(* Logix 5000 project; controller R1USB70001_CWRU_Scenario_Gen_20111116 vendor 1 type 14 code 54 rev 19.11; software revision 19.01; part 7 of 9 *)
(* tags used below, declared in another part *)
   EditScenario : EditScenarioPub;
   HMI : HMIPub;
   HMI_Intfc_Read_Buffer : DINT[40];
(* MainProgram, continued *)

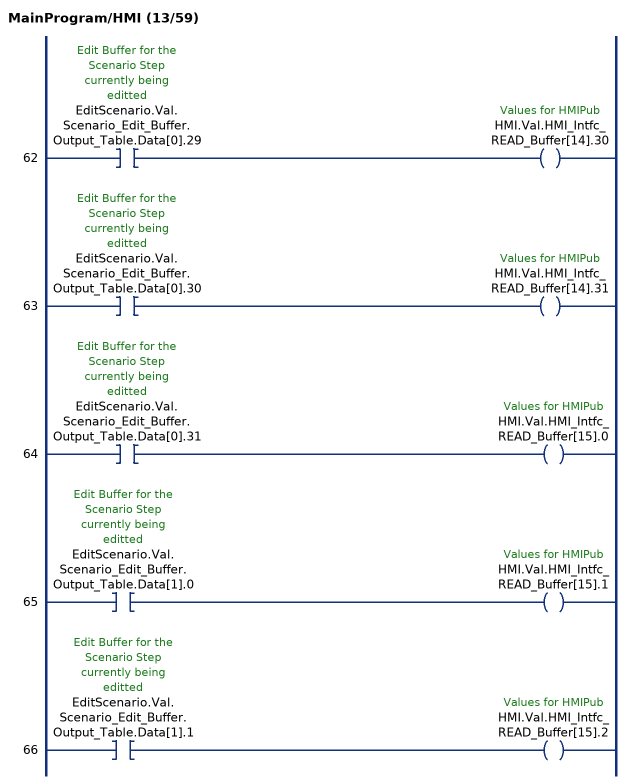
   62: XIC(EditScenario.Val.Scenario_Edit_Buffer.Output_Table.Data[0].29)OTE(HMI.Val.HMI_Intfc_READ_Buffer[14].30);
   63: XIC(EditScenario.Val.Scenario_Edit_Buffer.Output_Table.Data[0].30)OTE(HMI.Val.HMI_Intfc_READ_Buffer[14].31);
   64: XIC(EditScenario.Val.Scenario_Edit_Buffer.Output_Table.Data[0].31)OTE(HMI.Val.HMI_Intfc_READ_Buffer[15].0);
   65: XIC(EditScenario.Val.Scenario_Edit_Buffer.Output_Table.Data[1].0)OTE(HMI.Val.HMI_Intfc_READ_Buffer[15].1);
   66: XIC(EditScenario.Val.Scenario_Edit_Buffer.Output_Table.Data[1].1)OTE(HMI.Val.HMI_Intfc_READ_Buffer[15].2);
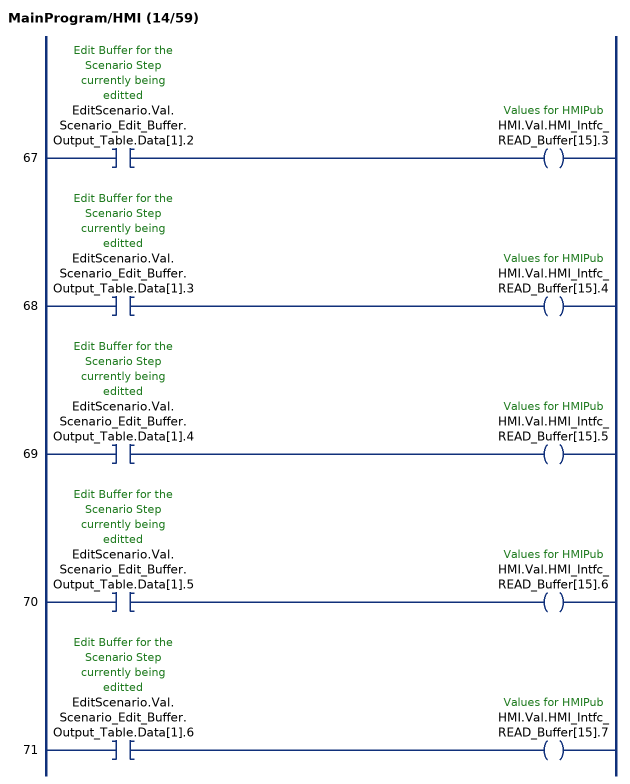
   67: XIC(EditScenario.Val.Scenario_Edit_Buffer.Output_Table.Data[1].2)OTE(HMI.Val.HMI_Intfc_READ_Buffer[15].3);
   68: XIC(EditScenario.Val.Scenario_Edit_Buffer.Output_Table.Data[1].3)OTE(HMI.Val.HMI_Intfc_READ_Buffer[15].4);
   69: XIC(EditScenario.Val.Scenario_Edit_Buffer.Output_Table.Data[1].4)OTE(HMI.Val.HMI_Intfc_READ_Buffer[15].5);
   70: XIC(EditScenario.Val.Scenario_Edit_Buffer.Output_Table.Data[1].5)OTE(HMI.Val.HMI_Intfc_READ_Buffer[15].6);
   71: XIC(EditScenario.Val.Scenario_Edit_Buffer.Output_Table.Data[1].6)OTE(HMI.Val.HMI_Intfc_READ_Buffer[15].7);
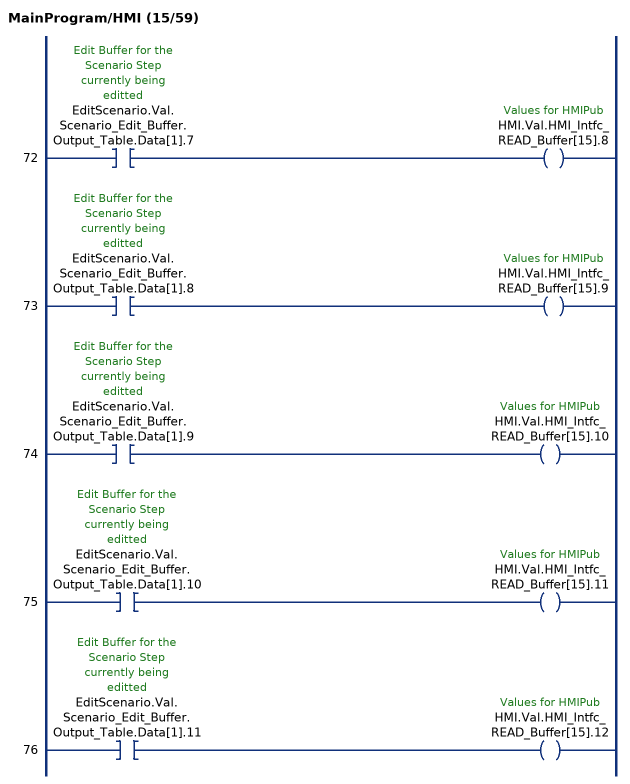
   72: XIC(EditScenario.Val.Scenario_Edit_Buffer.Output_Table.Data[1].7)OTE(HMI.Val.HMI_Intfc_READ_Buffer[15].8);
   73: XIC(EditScenario.Val.Scenario_Edit_Buffer.Output_Table.Data[1].8)OTE(HMI.Val.HMI_Intfc_READ_Buffer[15].9);
   74: XIC(EditScenario.Val.Scenario_Edit_Buffer.Output_Table.Data[1].9)OTE(HMI.Val.HMI_Intfc_READ_Buffer[15].10);
   75: XIC(EditScenario.Val.Scenario_Edit_Buffer.Output_Table.Data[1].10)OTE(HMI.Val.HMI_Intfc_READ_Buffer[15].11);
   76: XIC(EditScenario.Val.Scenario_Edit_Buffer.Output_Table.Data[1].11)OTE(HMI.Val.HMI_Intfc_READ_Buffer[15].12);
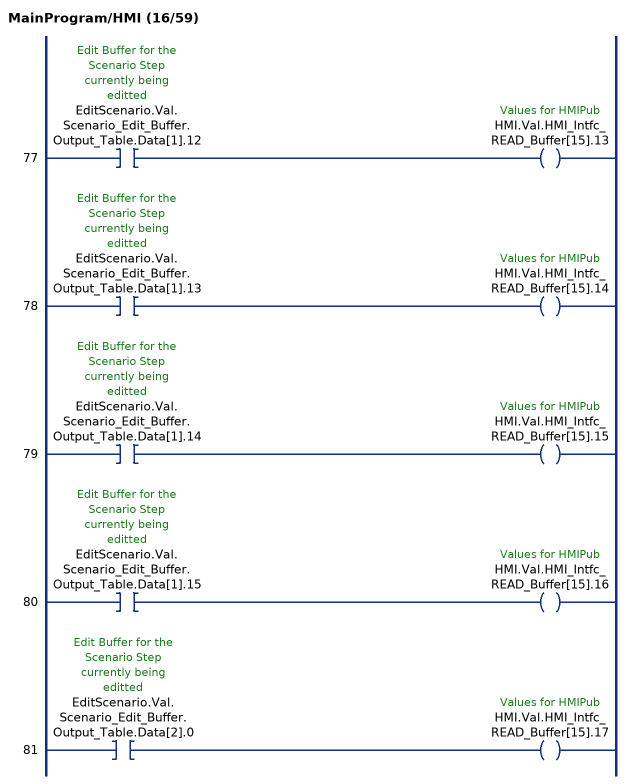
   77: XIC(EditScenario.Val.Scenario_Edit_Buffer.Output_Table.Data[1].12)OTE(HMI.Val.HMI_Intfc_READ_Buffer[15].13);
   78: XIC(EditScenario.Val.Scenario_Edit_Buffer.Output_Table.Data[1].13)OTE(HMI.Val.HMI_Intfc_READ_Buffer[15].14);
   79: XIC(EditScenario.Val.Scenario_Edit_Buffer.Output_Table.Data[1].14)OTE(HMI.Val.HMI_Intfc_READ_Buffer[15].15);
   80: XIC(EditScenario.Val.Scenario_Edit_Buffer.Output_Table.Data[1].15)OTE(HMI.Val.HMI_Intfc_READ_Buffer[15].16);
   81: XIC(EditScenario.Val.Scenario_Edit_Buffer.Output_Table.Data[2].0)OTE(HMI.Val.HMI_Intfc_READ_Buffer[15].17);
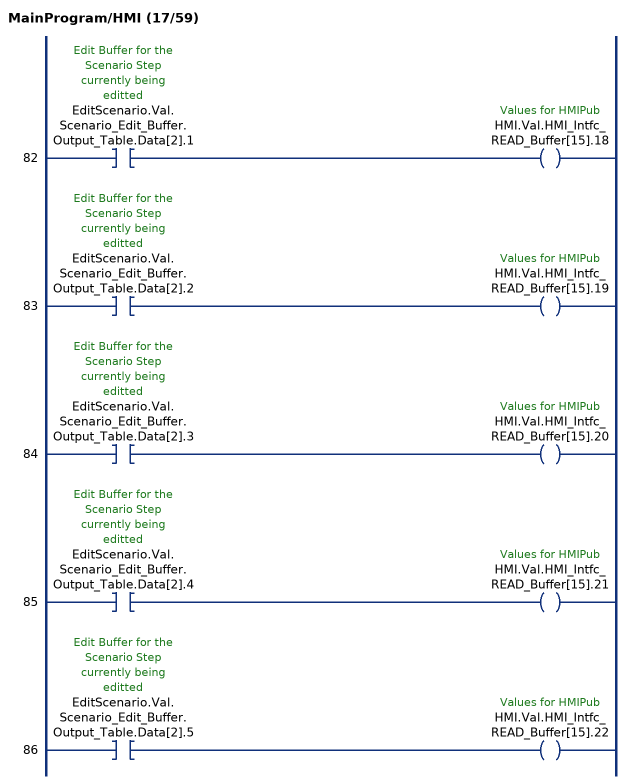
   82: XIC(EditScenario.Val.Scenario_Edit_Buffer.Output_Table.Data[2].1)OTE(HMI.Val.HMI_Intfc_READ_Buffer[15].18);
   83: XIC(EditScenario.Val.Scenario_Edit_Buffer.Output_Table.Data[2].2)OTE(HMI.Val.HMI_Intfc_READ_Buffer[15].19);
   84: XIC(EditScenario.Val.Scenario_Edit_Buffer.Output_Table.Data[2].3)OTE(HMI.Val.HMI_Intfc_READ_Buffer[15].20);
   85: XIC(EditScenario.Val.Scenario_Edit_Buffer.Output_Table.Data[2].4)OTE(HMI.Val.HMI_Intfc_READ_Buffer[15].21);
   86: XIC(EditScenario.Val.Scenario_Edit_Buffer.Output_Table.Data[2].5)OTE(HMI.Val.HMI_Intfc_READ_Buffer[15].22);
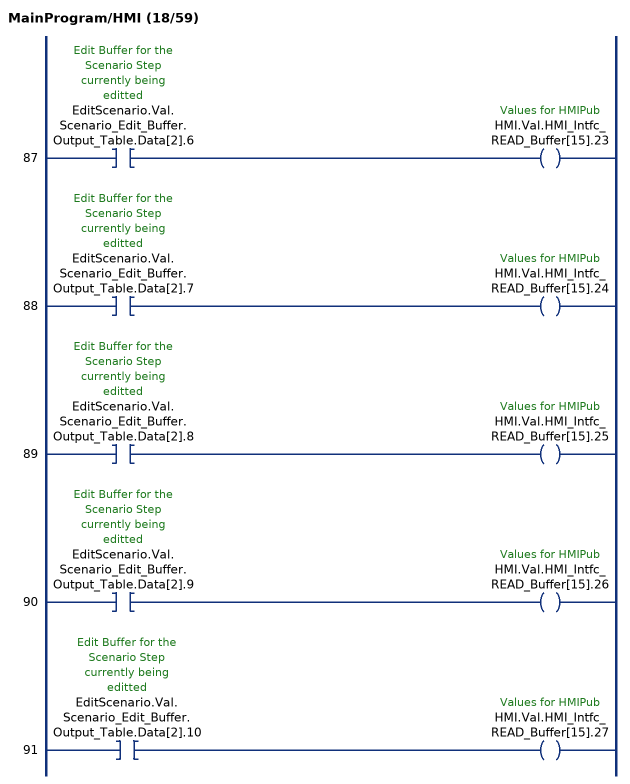
   87: XIC(EditScenario.Val.Scenario_Edit_Buffer.Output_Table.Data[2].6)OTE(HMI.Val.HMI_Intfc_READ_Buffer[15].23);
   88: XIC(EditScenario.Val.Scenario_Edit_Buffer.Output_Table.Data[2].7)OTE(HMI.Val.HMI_Intfc_READ_Buffer[15].24);
   89: XIC(EditScenario.Val.Scenario_Edit_Buffer.Output_Table.Data[2].8)OTE(HMI.Val.HMI_Intfc_READ_Buffer[15].25);
   90: XIC(EditScenario.Val.Scenario_Edit_Buffer.Output_Table.Data[2].9)OTE(HMI.Val.HMI_Intfc_READ_Buffer[15].26);
   91: XIC(EditScenario.Val.Scenario_Edit_Buffer.Output_Table.Data[2].10)OTE(HMI.Val.HMI_Intfc_READ_Buffer[15].27);
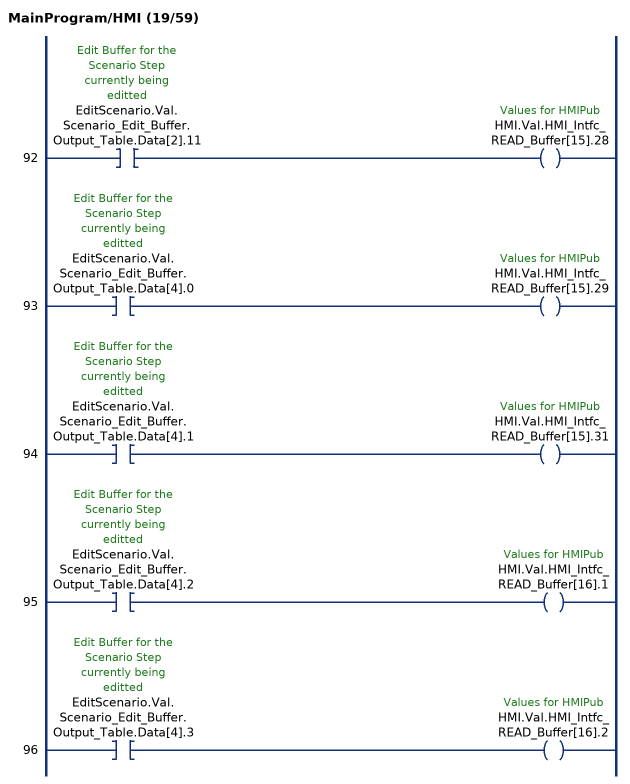
   92: XIC(EditScenario.Val.Scenario_Edit_Buffer.Output_Table.Data[2].11)OTE(HMI.Val.HMI_Intfc_READ_Buffer[15].28);
   93: XIC(EditScenario.Val.Scenario_Edit_Buffer.Output_Table.Data[4].0)OTE(HMI.Val.HMI_Intfc_READ_Buffer[15].29);
   94: XIC(EditScenario.Val.Scenario_Edit_Buffer.Output_Table.Data[4].1)OTE(HMI.Val.HMI_Intfc_READ_Buffer[15].31);
   95: XIC(EditScenario.Val.Scenario_Edit_Buffer.Output_Table.Data[4].2)OTE(HMI.Val.HMI_Intfc_READ_Buffer[16].1);
   96: XIC(EditScenario.Val.Scenario_Edit_Buffer.Output_Table.Data[4].3)OTE(HMI.Val.HMI_Intfc_READ_Buffer[16].2);
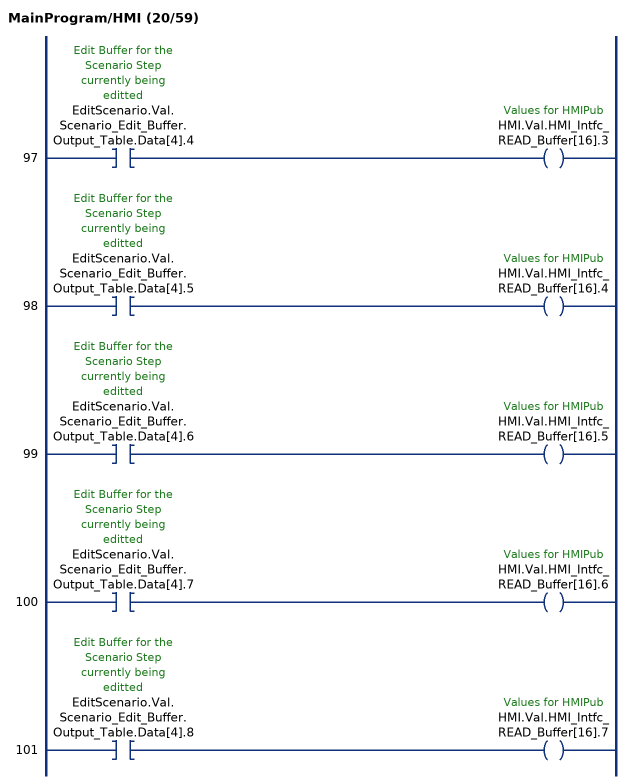
   97: XIC(EditScenario.Val.Scenario_Edit_Buffer.Output_Table.Data[4].4)OTE(HMI.Val.HMI_Intfc_READ_Buffer[16].3);
   98: XIC(EditScenario.Val.Scenario_Edit_Buffer.Output_Table.Data[4].5)OTE(HMI.Val.HMI_Intfc_READ_Buffer[16].4);
   99: XIC(EditScenario.Val.Scenario_Edit_Buffer.Output_Table.Data[4].6)OTE(HMI.Val.HMI_Intfc_READ_Buffer[16].5);
   100: XIC(EditScenario.Val.Scenario_Edit_Buffer.Output_Table.Data[4].7)OTE(HMI.Val.HMI_Intfc_READ_Buffer[16].6);
   101: XIC(EditScenario.Val.Scenario_Edit_Buffer.Output_Table.Data[4].8)OTE(HMI.Val.HMI_Intfc_READ_Buffer[16].7);
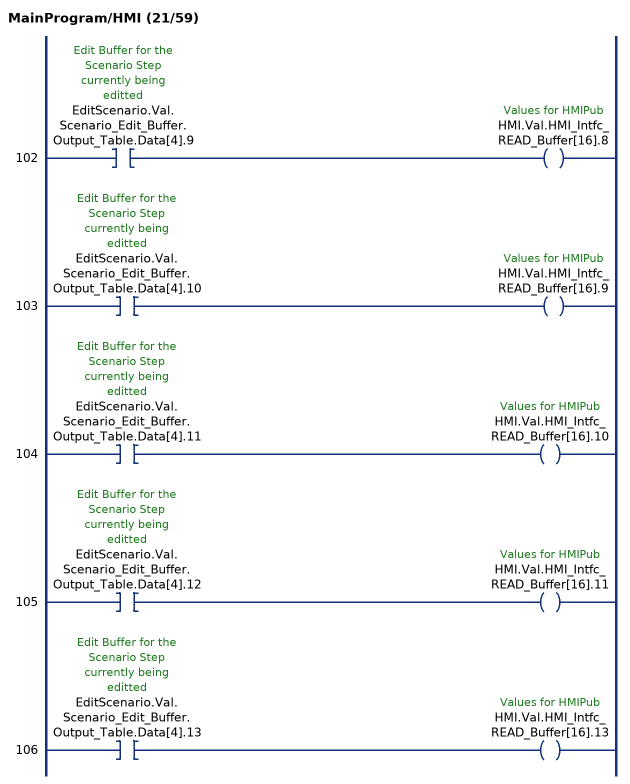
   102: XIC(EditScenario.Val.Scenario_Edit_Buffer.Output_Table.Data[4].9)OTE(HMI.Val.HMI_Intfc_READ_Buffer[16].8);
   103: XIC(EditScenario.Val.Scenario_Edit_Buffer.Output_Table.Data[4].10)OTE(HMI.Val.HMI_Intfc_READ_Buffer[16].9);
   104: XIC(EditScenario.Val.Scenario_Edit_Buffer.Output_Table.Data[4].11)OTE(HMI.Val.HMI_Intfc_READ_Buffer[16].10);
   105: XIC(EditScenario.Val.Scenario_Edit_Buffer.Output_Table.Data[4].12)OTE(HMI.Val.HMI_Intfc_READ_Buffer[16].11);
   106: XIC(EditScenario.Val.Scenario_Edit_Buffer.Output_Table.Data[4].13)OTE(HMI.Val.HMI_Intfc_READ_Buffer[16].13);
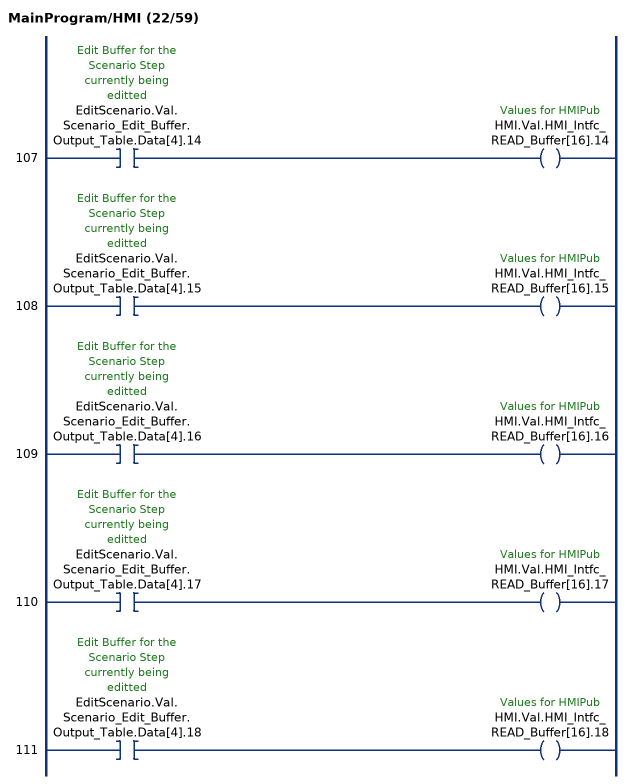
   107: XIC(EditScenario.Val.Scenario_Edit_Buffer.Output_Table.Data[4].14)OTE(HMI.Val.HMI_Intfc_READ_Buffer[16].14);
   108: XIC(EditScenario.Val.Scenario_Edit_Buffer.Output_Table.Data[4].15)OTE(HMI.Val.HMI_Intfc_READ_Buffer[16].15);
   109: XIC(EditScenario.Val.Scenario_Edit_Buffer.Output_Table.Data[4].16)OTE(HMI.Val.HMI_Intfc_READ_Buffer[16].16);
   110: XIC(EditScenario.Val.Scenario_Edit_Buffer.Output_Table.Data[4].17)OTE(HMI.Val.HMI_Intfc_READ_Buffer[16].17);
   111: XIC(EditScenario.Val.Scenario_Edit_Buffer.Output_Table.Data[4].18)OTE(HMI.Val.HMI_Intfc_READ_Buffer[16].18);
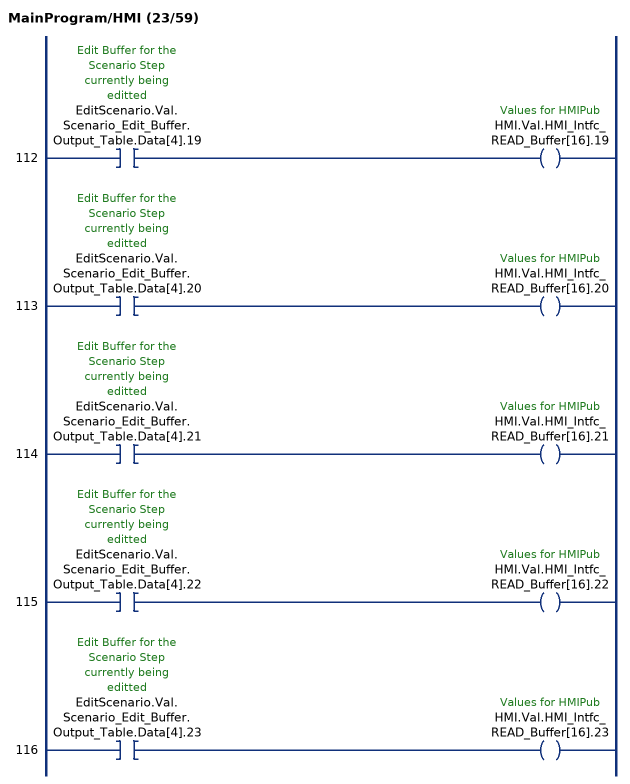
   112: XIC(EditScenario.Val.Scenario_Edit_Buffer.Output_Table.Data[4].19)OTE(HMI.Val.HMI_Intfc_READ_Buffer[16].19);
   113: XIC(EditScenario.Val.Scenario_Edit_Buffer.Output_Table.Data[4].20)OTE(HMI.Val.HMI_Intfc_READ_Buffer[16].20);
   114: XIC(EditScenario.Val.Scenario_Edit_Buffer.Output_Table.Data[4].21)OTE(HMI.Val.HMI_Intfc_READ_Buffer[16].21);
   115: XIC(EditScenario.Val.Scenario_Edit_Buffer.Output_Table.Data[4].22)OTE(HMI.Val.HMI_Intfc_READ_Buffer[16].22);
   116: XIC(EditScenario.Val.Scenario_Edit_Buffer.Output_Table.Data[4].23)OTE(HMI.Val.HMI_Intfc_READ_Buffer[16].23);
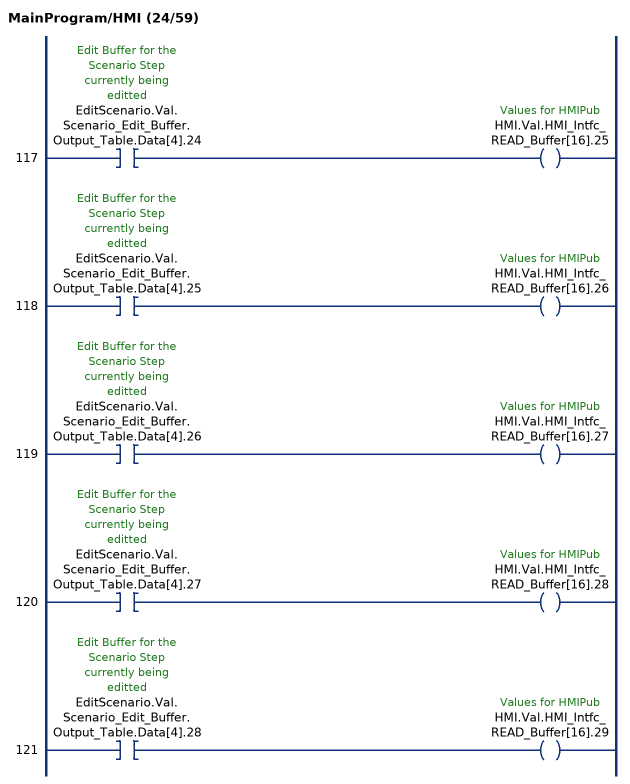
   117: XIC(EditScenario.Val.Scenario_Edit_Buffer.Output_Table.Data[4].24)OTE(HMI.Val.HMI_Intfc_READ_Buffer[16].25);
   118: XIC(EditScenario.Val.Scenario_Edit_Buffer.Output_Table.Data[4].25)OTE(HMI.Val.HMI_Intfc_READ_Buffer[16].26);
   119: XIC(EditScenario.Val.Scenario_Edit_Buffer.Output_Table.Data[4].26)OTE(HMI.Val.HMI_Intfc_READ_Buffer[16].27);
   120: XIC(EditScenario.Val.Scenario_Edit_Buffer.Output_Table.Data[4].27)OTE(HMI.Val.HMI_Intfc_READ_Buffer[16].28);
   121: XIC(EditScenario.Val.Scenario_Edit_Buffer.Output_Table.Data[4].28)OTE(HMI.Val.HMI_Intfc_READ_Buffer[16].29);
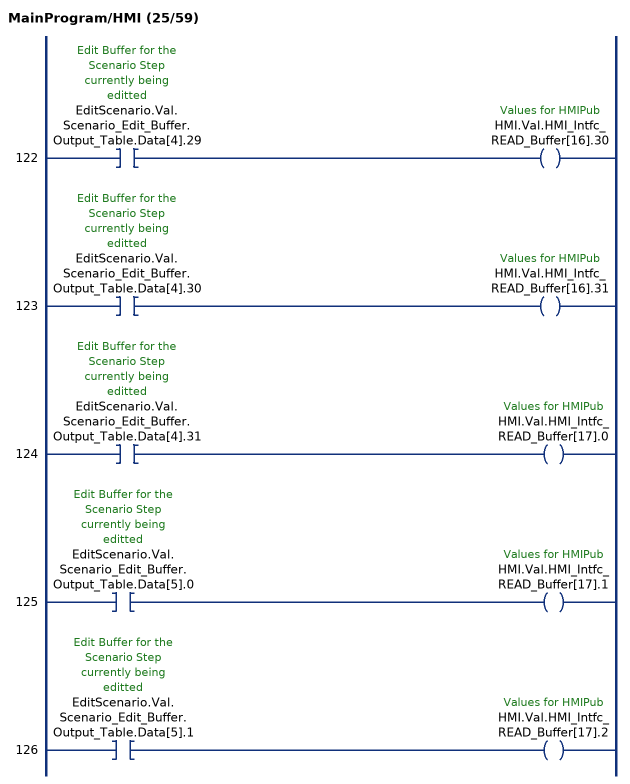
   122: XIC(EditScenario.Val.Scenario_Edit_Buffer.Output_Table.Data[4].29)OTE(HMI.Val.HMI_Intfc_READ_Buffer[16].30);
   123: XIC(EditScenario.Val.Scenario_Edit_Buffer.Output_Table.Data[4].30)OTE(HMI.Val.HMI_Intfc_READ_Buffer[16].31);
   124: XIC(EditScenario.Val.Scenario_Edit_Buffer.Output_Table.Data[4].31)OTE(HMI.Val.HMI_Intfc_READ_Buffer[17].0);
   125: XIC(EditScenario.Val.Scenario_Edit_Buffer.Output_Table.Data[5].0)OTE(HMI.Val.HMI_Intfc_READ_Buffer[17].1);
   126: XIC(EditScenario.Val.Scenario_Edit_Buffer.Output_Table.Data[5].1)OTE(HMI.Val.HMI_Intfc_READ_Buffer[17].2);
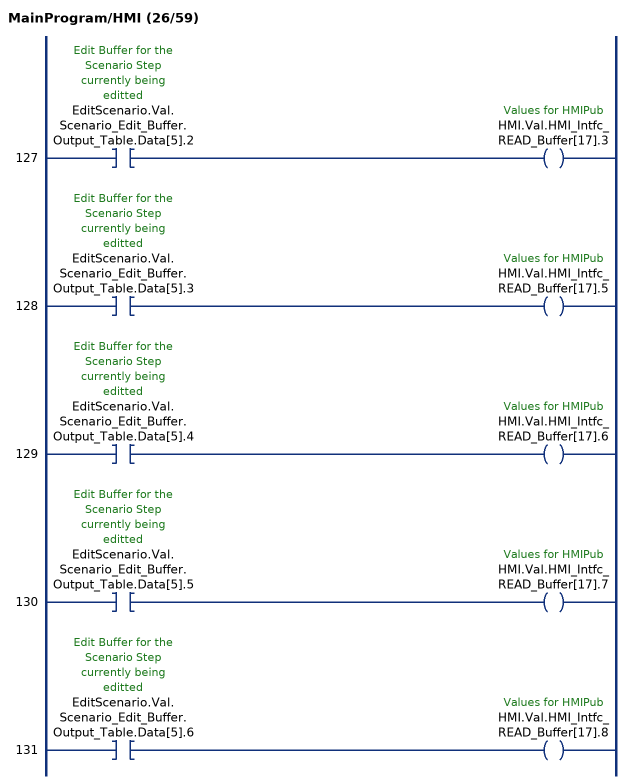
   127: XIC(EditScenario.Val.Scenario_Edit_Buffer.Output_Table.Data[5].2)OTE(HMI.Val.HMI_Intfc_READ_Buffer[17].3);
   128: XIC(EditScenario.Val.Scenario_Edit_Buffer.Output_Table.Data[5].3)OTE(HMI.Val.HMI_Intfc_READ_Buffer[17].5);
   129: XIC(EditScenario.Val.Scenario_Edit_Buffer.Output_Table.Data[5].4)OTE(HMI.Val.HMI_Intfc_READ_Buffer[17].6);
   130: XIC(EditScenario.Val.Scenario_Edit_Buffer.Output_Table.Data[5].5)OTE(HMI.Val.HMI_Intfc_READ_Buffer[17].7);
   131: XIC(EditScenario.Val.Scenario_Edit_Buffer.Output_Table.Data[5].6)OTE(HMI.Val.HMI_Intfc_READ_Buffer[17].8);
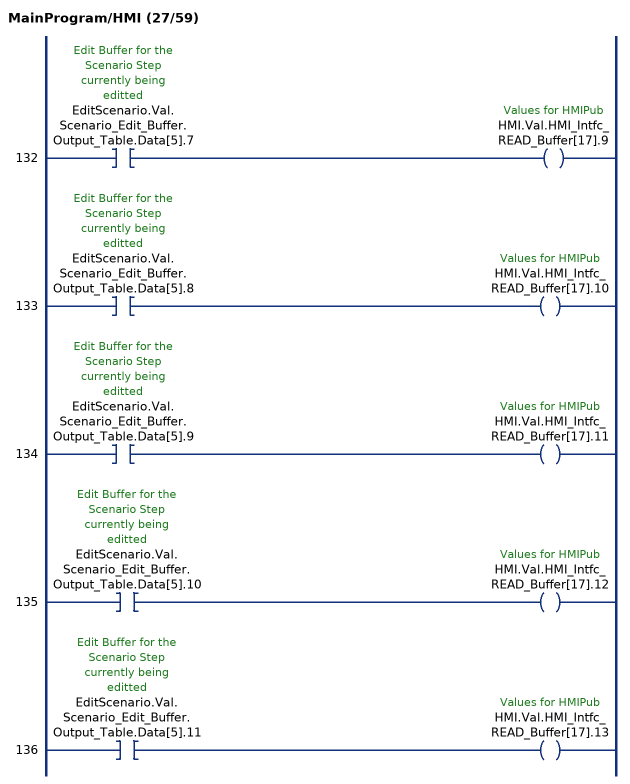
   132: XIC(EditScenario.Val.Scenario_Edit_Buffer.Output_Table.Data[5].7)OTE(HMI.Val.HMI_Intfc_READ_Buffer[17].9);
   133: XIC(EditScenario.Val.Scenario_Edit_Buffer.Output_Table.Data[5].8)OTE(HMI.Val.HMI_Intfc_READ_Buffer[17].10);
   134: XIC(EditScenario.Val.Scenario_Edit_Buffer.Output_Table.Data[5].9)OTE(HMI.Val.HMI_Intfc_READ_Buffer[17].11);
   135: XIC(EditScenario.Val.Scenario_Edit_Buffer.Output_Table.Data[5].10)OTE(HMI.Val.HMI_Intfc_READ_Buffer[17].12);
   136: XIC(EditScenario.Val.Scenario_Edit_Buffer.Output_Table.Data[5].11)OTE(HMI.Val.HMI_Intfc_READ_Buffer[17].13);
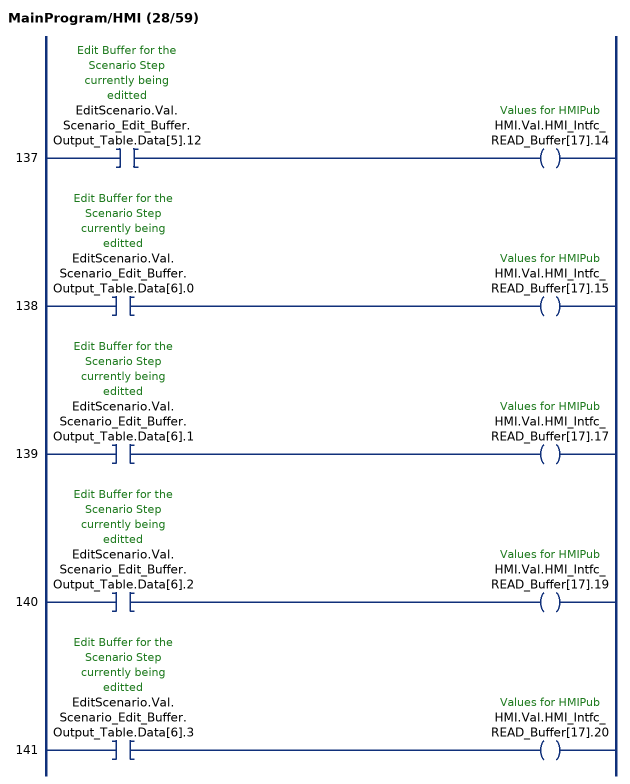
   137: XIC(EditScenario.Val.Scenario_Edit_Buffer.Output_Table.Data[5].12)OTE(HMI.Val.HMI_Intfc_READ_Buffer[17].14);
   138: XIC(EditScenario.Val.Scenario_Edit_Buffer.Output_Table.Data[6].0)OTE(HMI.Val.HMI_Intfc_READ_Buffer[17].15);
   139: XIC(EditScenario.Val.Scenario_Edit_Buffer.Output_Table.Data[6].1)OTE(HMI.Val.HMI_Intfc_READ_Buffer[17].17);
   140: XIC(EditScenario.Val.Scenario_Edit_Buffer.Output_Table.Data[6].2)OTE(HMI.Val.HMI_Intfc_READ_Buffer[17].19);
   141: XIC(EditScenario.Val.Scenario_Edit_Buffer.Output_Table.Data[6].3)OTE(HMI.Val.HMI_Intfc_READ_Buffer[17].20);
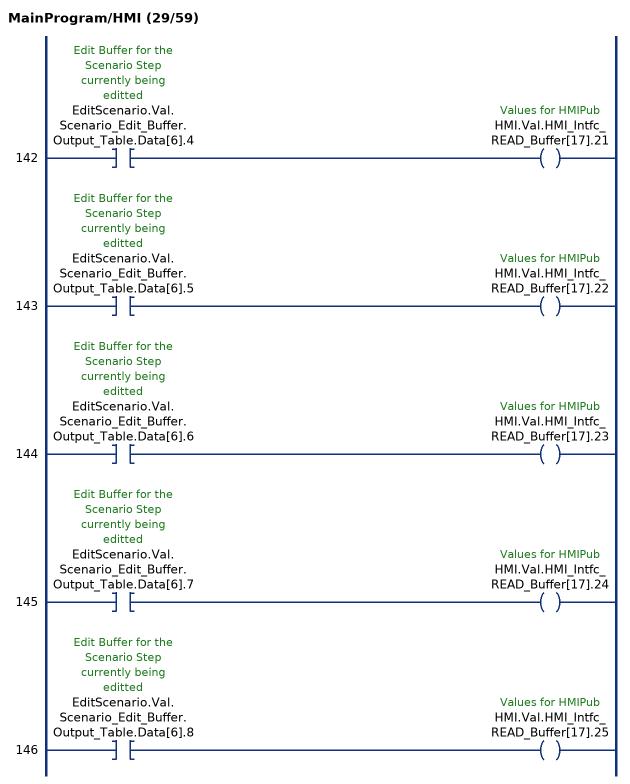
   142: XIC(EditScenario.Val.Scenario_Edit_Buffer.Output_Table.Data[6].4)OTE(HMI.Val.HMI_Intfc_READ_Buffer[17].21);
   143: XIC(EditScenario.Val.Scenario_Edit_Buffer.Output_Table.Data[6].5)OTE(HMI.Val.HMI_Intfc_READ_Buffer[17].22);
   144: XIC(EditScenario.Val.Scenario_Edit_Buffer.Output_Table.Data[6].6)OTE(HMI.Val.HMI_Intfc_READ_Buffer[17].23);
   145: XIC(EditScenario.Val.Scenario_Edit_Buffer.Output_Table.Data[6].7)OTE(HMI.Val.HMI_Intfc_READ_Buffer[17].24);
   146: XIC(EditScenario.Val.Scenario_Edit_Buffer.Output_Table.Data[6].8)OTE(HMI.Val.HMI_Intfc_READ_Buffer[17].25);
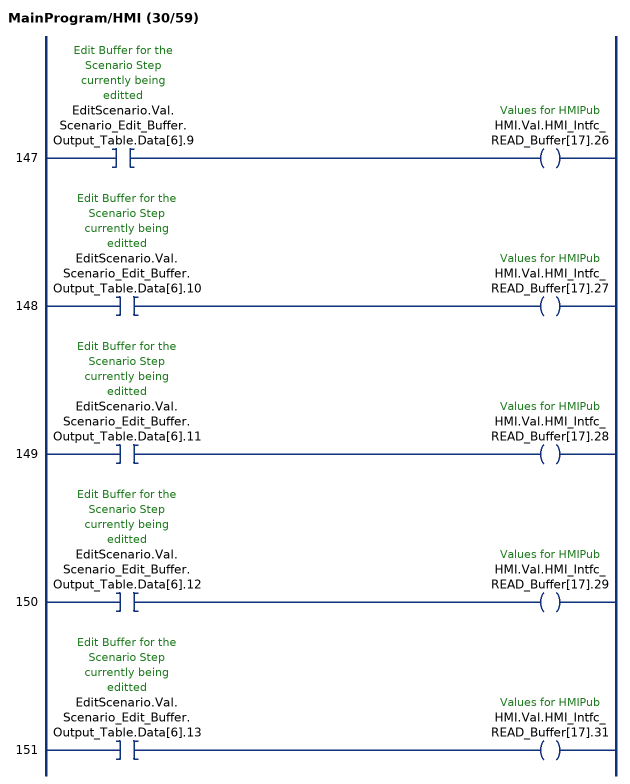
   147: XIC(EditScenario.Val.Scenario_Edit_Buffer.Output_Table.Data[6].9)OTE(HMI.Val.HMI_Intfc_READ_Buffer[17].26);
   148: XIC(EditScenario.Val.Scenario_Edit_Buffer.Output_Table.Data[6].10)OTE(HMI.Val.HMI_Intfc_READ_Buffer[17].27);
   149: XIC(EditScenario.Val.Scenario_Edit_Buffer.Output_Table.Data[6].11)OTE(HMI.Val.HMI_Intfc_READ_Buffer[17].28);
   150: XIC(EditScenario.Val.Scenario_Edit_Buffer.Output_Table.Data[6].12)OTE(HMI.Val.HMI_Intfc_READ_Buffer[17].29);
   151: XIC(EditScenario.Val.Scenario_Edit_Buffer.Output_Table.Data[6].13)OTE(HMI.Val.HMI_Intfc_READ_Buffer[17].31);
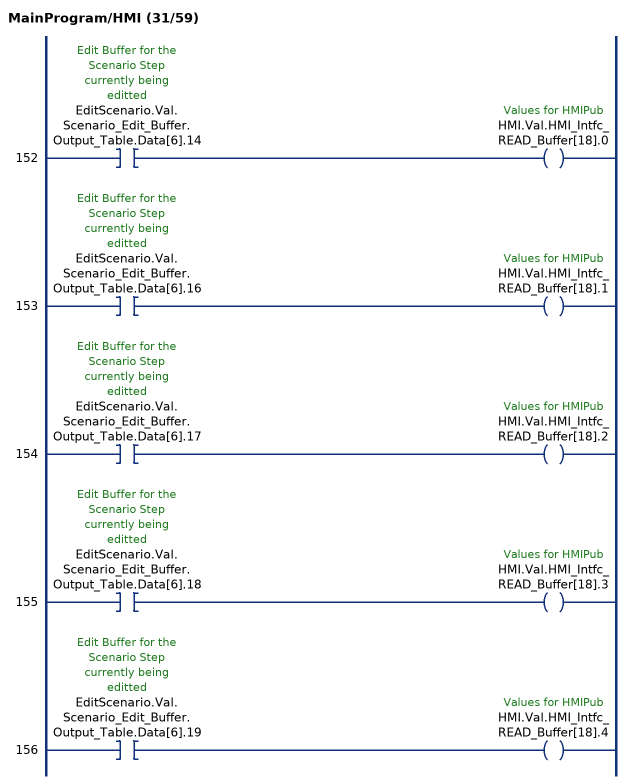
   152: XIC(EditScenario.Val.Scenario_Edit_Buffer.Output_Table.Data[6].14)OTE(HMI.Val.HMI_Intfc_READ_Buffer[18].0);
   153: XIC(EditScenario.Val.Scenario_Edit_Buffer.Output_Table.Data[6].16)OTE(HMI.Val.HMI_Intfc_READ_Buffer[18].1);
   154: XIC(EditScenario.Val.Scenario_Edit_Buffer.Output_Table.Data[6].17)OTE(HMI.Val.HMI_Intfc_READ_Buffer[18].2);
   155: XIC(EditScenario.Val.Scenario_Edit_Buffer.Output_Table.Data[6].18)OTE(HMI.Val.HMI_Intfc_READ_Buffer[18].3);
   156: XIC(EditScenario.Val.Scenario_Edit_Buffer.Output_Table.Data[6].19)OTE(HMI.Val.HMI_Intfc_READ_Buffer[18].4);
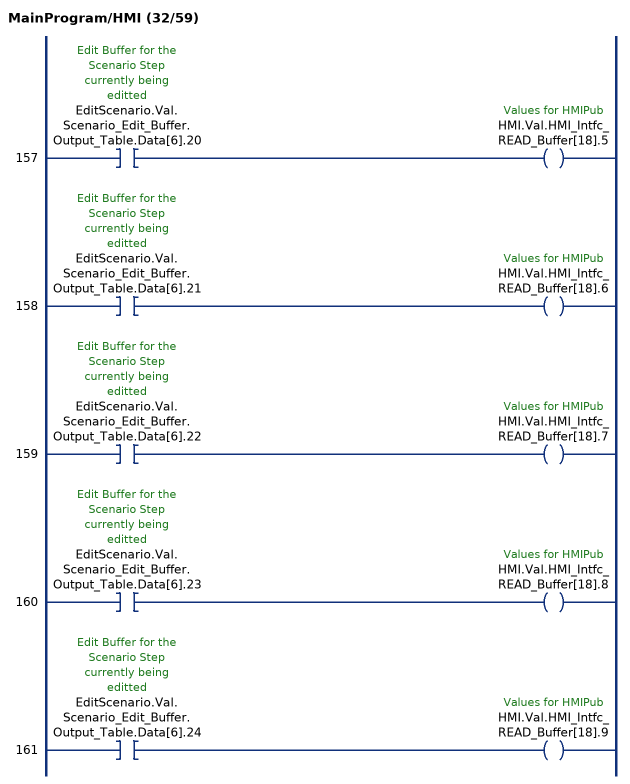
   157: XIC(EditScenario.Val.Scenario_Edit_Buffer.Output_Table.Data[6].20)OTE(HMI.Val.HMI_Intfc_READ_Buffer[18].5);
   158: XIC(EditScenario.Val.Scenario_Edit_Buffer.Output_Table.Data[6].21)OTE(HMI.Val.HMI_Intfc_READ_Buffer[18].6);
   159: XIC(EditScenario.Val.Scenario_Edit_Buffer.Output_Table.Data[6].22)OTE(HMI.Val.HMI_Intfc_READ_Buffer[18].7);
   160: XIC(EditScenario.Val.Scenario_Edit_Buffer.Output_Table.Data[6].23)OTE(HMI.Val.HMI_Intfc_READ_Buffer[18].8);
   161: XIC(EditScenario.Val.Scenario_Edit_Buffer.Output_Table.Data[6].24)OTE(HMI.Val.HMI_Intfc_READ_Buffer[18].9);
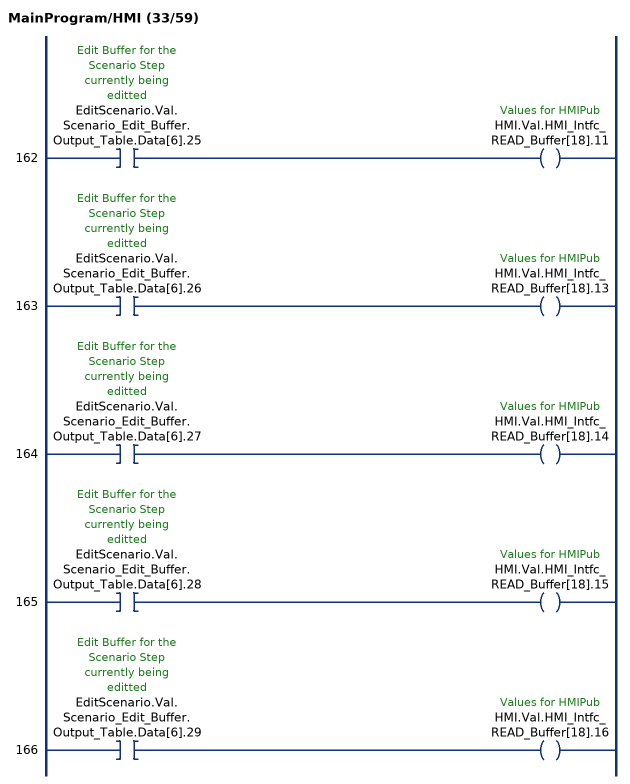
   162: XIC(EditScenario.Val.Scenario_Edit_Buffer.Output_Table.Data[6].25)OTE(HMI.Val.HMI_Intfc_READ_Buffer[18].11);
   163: XIC(EditScenario.Val.Scenario_Edit_Buffer.Output_Table.Data[6].26)OTE(HMI.Val.HMI_Intfc_READ_Buffer[18].13);
   164: XIC(EditScenario.Val.Scenario_Edit_Buffer.Output_Table.Data[6].27)OTE(HMI.Val.HMI_Intfc_READ_Buffer[18].14);
   165: XIC(EditScenario.Val.Scenario_Edit_Buffer.Output_Table.Data[6].28)OTE(HMI.Val.HMI_Intfc_READ_Buffer[18].15);
   166: XIC(EditScenario.Val.Scenario_Edit_Buffer.Output_Table.Data[6].29)OTE(HMI.Val.HMI_Intfc_READ_Buffer[18].16);
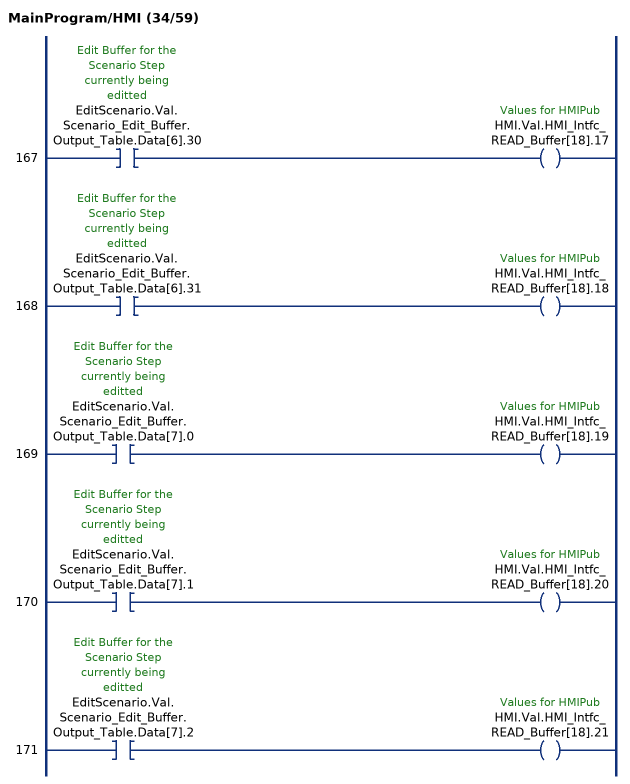
   167: XIC(EditScenario.Val.Scenario_Edit_Buffer.Output_Table.Data[6].30)OTE(HMI.Val.HMI_Intfc_READ_Buffer[18].17);
   168: XIC(EditScenario.Val.Scenario_Edit_Buffer.Output_Table.Data[6].31)OTE(HMI.Val.HMI_Intfc_READ_Buffer[18].18);
   169: XIC(EditScenario.Val.Scenario_Edit_Buffer.Output_Table.Data[7].0)OTE(HMI.Val.HMI_Intfc_READ_Buffer[18].19);
   170: XIC(EditScenario.Val.Scenario_Edit_Buffer.Output_Table.Data[7].1)OTE(HMI.Val.HMI_Intfc_READ_Buffer[18].20);
   171: XIC(EditScenario.Val.Scenario_Edit_Buffer.Output_Table.Data[7].2)OTE(HMI.Val.HMI_Intfc_READ_Buffer[18].21);
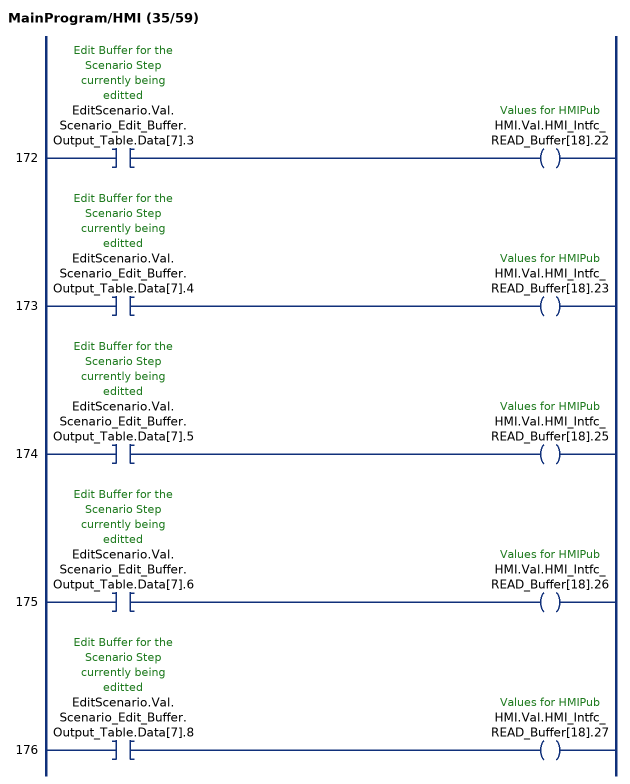
   172: XIC(EditScenario.Val.Scenario_Edit_Buffer.Output_Table.Data[7].3)OTE(HMI.Val.HMI_Intfc_READ_Buffer[18].22);
   173: XIC(EditScenario.Val.Scenario_Edit_Buffer.Output_Table.Data[7].4)OTE(HMI.Val.HMI_Intfc_READ_Buffer[18].23);
   174: XIC(EditScenario.Val.Scenario_Edit_Buffer.Output_Table.Data[7].5)OTE(HMI.Val.HMI_Intfc_READ_Buffer[18].25);
   175: XIC(EditScenario.Val.Scenario_Edit_Buffer.Output_Table.Data[7].6)OTE(HMI.Val.HMI_Intfc_READ_Buffer[18].26);
   176: XIC(EditScenario.Val.Scenario_Edit_Buffer.Output_Table.Data[7].8)OTE(HMI.Val.HMI_Intfc_READ_Buffer[18].27);
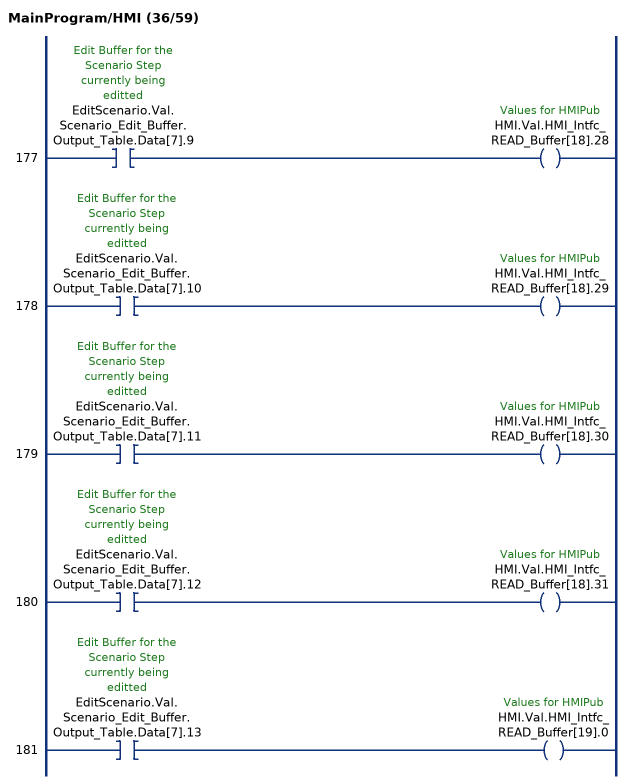
   177: XIC(EditScenario.Val.Scenario_Edit_Buffer.Output_Table.Data[7].9)OTE(HMI.Val.HMI_Intfc_READ_Buffer[18].28);
   178: XIC(EditScenario.Val.Scenario_Edit_Buffer.Output_Table.Data[7].10)OTE(HMI.Val.HMI_Intfc_READ_Buffer[18].29);
   179: XIC(EditScenario.Val.Scenario_Edit_Buffer.Output_Table.Data[7].11)OTE(HMI.Val.HMI_Intfc_READ_Buffer[18].30);
   180: XIC(EditScenario.Val.Scenario_Edit_Buffer.Output_Table.Data[7].12)OTE(HMI.Val.HMI_Intfc_READ_Buffer[18].31);
   181: XIC(EditScenario.Val.Scenario_Edit_Buffer.Output_Table.Data[7].13)OTE(HMI.Val.HMI_Intfc_READ_Buffer[19].0);
